// TIA Portal V17 export
// export: Created 2024-08-20T13:26:11.7387081Z, ExportSetting WithDefaults, DisplayName Totally Integrated Automation Portal, DisplayVersion V17 Update 4, DisplayName TIA Portal Openness, DisplayVersion V17 Update 4, DisplayName TIA Portal Version Control Interface, DisplayVersion V17, DisplayName STEP 7 Professional, DisplayVersion V17 Update 4, DisplayName STEP 7 Safety, DisplayVersion V17, DisplayName WinCC Advanced, DisplayVersion V17 Update 4
DATA_BLOCK "PID"   // DB307
{ S7_Optimized_Access := 'FALSE' }
VERSION : 0.1
// stored: AutoNumber false, DBAccessibleFromOPCUA true, IsOnlyStoredInLoadMemory false, IsWriteProtectedInAS false
   VAR RETAIN
      "PID-EEEB-D" : Real;   // Ajuste derivativo PID elevatória de esgoto bruto
      "PID-EEEB-P" : Real;   // Ajuste proporcional PID elevatória de esgoto bruto
      "PID-EEEB-I" : Real;   // Ajuste integral PID elevatória de esgoto bruto
      "PID-EEEB-MIN" : Real;   // Ajuste mínimo PID elevatória de esgoto bruto
      "PID-EEEB-MAX" : Real;   // Ajuste máximo PID elevatória de esgoto bruto
      "PID-EEEB-DB" : Real;   // Banda morta PID elevatória de esgoto bruto
      "PID-EEEB-SPM" : Real;   // Setpoint manual
      "VA-PID-EEEB" : Real;   // Variável atuada PID elevatória de esgoto bruto
      "PID-EEEB-VR" : Real;   // Valor Relativo do PID
      AUX_CALC : Array[0..10] of Real;
   END_VAR
BEGIN
END_DATA_BLOCK
